FUNCTION_BLOCK EventCounter (* Basic Function Block Type *)
  (* Standard: 61499-2 *)
  (* Version 0.0, 11/22/2016, chivdan, nxtControl GmbH, Template *)
  PACKAGE Main;
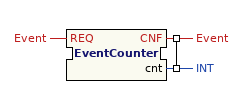
  EVENT_INPUT
    REQ; (* Normal Execution Request *)
  END_EVENT
  EVENT_OUTPUT
    CNF WITH cnt; (* Execution Confirmation *)
  END_EVENT
  VAR_OUTPUT
    cnt : INT := 0; (* Output event qualifier *)
  END_VAR
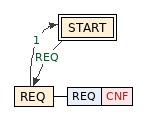
  EC_STATES
    START; (* Initial State *)
    REQ : REQ -> CNF; (* Normal execution *)
  END_STATES
  EC_TRANSITIONS
    START TO REQ := REQ;
    REQ TO START := 1;
  END_TRANSITIONS
  ALGORITHM INIT IN ST: (* Initialization algorithm *)
;
  END_ALGORITHM
  ALGORITHM REQ IN ST: (* Normally executed algorithm *)
;
cnt:=cnt+1;
  END_ALGORITHM
END_FUNCTION_BLOCK
